FUNCTION NmSetNameField
  (* Standard: 61499-1 *)
  (* Version 1.0, 2025-09-04, franz *)
  PACKAGE isobus;
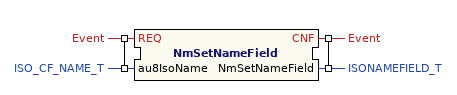
  EVENT_INPUT
    REQ WITH au8IsoName;
  END_EVENT
  EVENT_OUTPUT
    CNF WITH NmSetNameField;
  END_EVENT
  VAR_INPUT
    au8IsoName : isobus::ISO_CF_NAME_T;
  END_VAR
  VAR_OUTPUT
    NmSetNameField : ISONAMEFIELD_T;
  END_VAR
  BODY IN ST:
PACKAGE isobus;

FUNCTION NmSetNameField : ISONAMEFIELD_T
VAR_INPUT
	au8IsoName : ISO_CF_NAME_T;
END_VAR

// ISO NAME fields are 8 bytes long (0 to 7)
// The bits are assigned to the structured type ISONAMEFIELD_T
// Byte 7
NmSetNameField.bSelfConf := ((au8IsoName.data[7] AND WORD#16#80) = WORD#16#80);
NmSetNameField.bIndGroup := SHL(SHR(au8IsoName.data[7], SINT#4), SINT#1) AND BYTE#16#07;
NmSetNameField.bDevClassInst := au8IsoName.data[7] AND BYTE#16#0F;

// Byte 6
NmSetNameField.bDevClass := SHR(au8IsoName.data[6], SINT#1) AND BYTE#16#7F;
NmSetNameField.bReserved := ((au8IsoName.data[6] AND BYTE#16#01) = BYTE#16#01);

// Byte 5
NmSetNameField.bFunction := au8IsoName.data[5];

// Byte 4
NmSetNameField.bFunctionInst := SHR(au8IsoName.data[4], SINT#5) AND BYTE#16#1F;
NmSetNameField.bEcuInstance := au8IsoName.data[4] AND BYTE#16#1F;

// Bytes 2, 3 for Manufacturer Code
NmSetNameField.wManufCode := SHL(BYTE_TO_WORD(au8IsoName.data[3]), SINT#3)
	OR SHR(BYTE_TO_WORD(au8IsoName.data[2] AND BYTE#16#E0), SINT#5);

// Bytes 0, 1, 2 for Identity Number
NmSetNameField.dwIdentNumb := SHL(BYTE_TO_DWORD(au8IsoName.data[2] AND BYTE#16#1F), SINT#16)
	OR SHL(BYTE_TO_DWORD(au8IsoName.data[1]), SINT#8) OR BYTE_TO_DWORD(au8IsoName.data[0]);

END_FUNCTION
  END_BODY
END_FUNCTION
